(* CODESYS project FU_bBitSet.xml

Project tree, tasks and I/O mapping:
  function FU_bBitSet [ST]
*)

// FU_bBitSet
//This function sets the bit value from a variable
// |**Version**|**Author**| **Date** |**Changes**                                                                                                            |
// | 1         | NSN      | 11-01-19 | Creation                                                                                                              |
FUNCTION FU_bBitSet : BOOL
VAR_IN_OUT
	bVar	:BYTE;		//The value to work with
END_VAR
VAR_INPUT
	bIndex	:BYTE;		//Which bit to get
	xVal	:BOOL;		//What to set the bit to
END_VAR

bVar		:=		(bVar AND NOT(SHL(TO_BYTE(1),bIndex))) OR (SHL(TO_BYTE(xVal),bIndex));

END_FUNCTION
